TYPE s_gm_rotaryPos :
STRUCT
	origin	: LREAL;
	pickUp	: LREAL;
	set		: LREAL;
	remove  : LREAL;
END_STRUCT
END_TYPE

(* stored: Version 1.1.0.1, ProductVersion 3.1.4024.11
   DUT s_gm_rotaryPos: Id {2a5cfd23-108b-4e9c-892a-04126b17c814} *)
